// TIA Portal V20 export
TYPE "typeAxisIntlockAll"
// stored: Access Published, Namespace LER
   STRUCT
      Home { S7_SetPoint := 'True'} : "LER.typeAxisHomeCondition";
      Jog { S7_SetPoint := 'True'} : "LER.typeAxisJogCondition";
      Position { S7_SetPoint := 'True'} : "LER.typeAxisPositionCondition";
   END_STRUCT;
END_TYPE
